FUNCTION_BLOCK FB_XOR2 (* Composite XOR Function Block Type *)
  (* Standard: 61499-2 *)
  (* Version 0.0, 2004-06-07, JHC, HUT *)
  (* Compiler header: package fb.rt.student; import fb.rt.math.*; *)
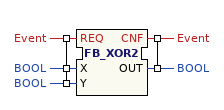
  EVENT_INPUT
    REQ WITH X, Y; (* Normal Execution Request *)
  END_EVENT
  EVENT_OUTPUT
    CNF WITH OUT; (* Execution Confirmation *)
  END_EVENT
  VAR_INPUT
    X : BOOL;
    Y : BOOL;
  END_VAR
  VAR_OUTPUT
    OUT : BOOL; (* X XOR Y *)
  END_VAR
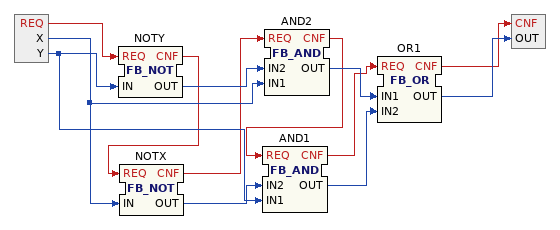
  FBS
    AND1 : FB_AND;
    AND2 : FB_AND;
    OR1 : FB_OR;
    NOTX : FB_NOT;
    NOTY : FB_NOT;
  END_FBS
  EVENT_CONNECTIONS
    REQ TO NOTY.REQ;
    NOTX.CNF TO AND2.REQ;
    AND2.CNF TO AND1.REQ;
    AND1.CNF TO OR1.REQ;
    NOTY.CNF TO NOTX.REQ;
    OR1.CNF TO CNF;
  END_CONNECTIONS
  DATA_CONNECTIONS
    AND2.OUT TO OR1.IN1;
    AND1.OUT TO OR1.IN2;
    NOTY.OUT TO AND2.IN2;
    NOTX.OUT TO AND1.IN2;
    Y TO NOTY.IN;
    X TO NOTX.IN;
    X TO AND2.IN1;
    Y TO AND1.IN1;
    OR1.OUT TO OUT;
  END_CONNECTIONS
END_FUNCTION_BLOCK
